(* CoDeSys 2.3 export: GLOBAL_VARIABLES.EXP *)

(* Global variable list: Global_Variables *)
VAR_GLOBAL
	AlwaysOne : BOOL := TRUE ;
END_VAR
